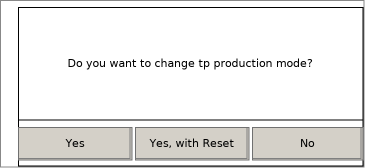
VISUALIZATION VIS_TemplateToProduction  // 365x168
VAR_IN_OUT
	stChangeIntoProduction	: ST_ChangeIntoProduction;
END_VAR
    Rectangle (18,9 345x157)
    Rectangle (18,7 345x113), "Do you want to change tp production mode?"
    Button (18,127 114x33), "Yes"
        tap stChangeIntoProduction.bYes
    Button (135,127 114x33), "Yes, with Reset"
        tap stChangeIntoProduction.bYesReset
    Button (252,127 111x33), "No"
        tap stChangeIntoProduction.bNo
END_VISUALIZATION

(* stored: Version 1.1.0.1, ProductVersion 3.1.4024.12
   Visu VIS_TemplateToProduction: Id {8935c84a-1028-477b-9d9f-fc5c2ff3fe77} *)
